FUNCTION F_DcToExt : T_DCTIME64  // Converts a DC time to a TAI-like absolute time expressed in T_DCTIME64 format.
VAR_INPUT
	dcTime: T_DCTIME64;  // 64-bit DC time.
END_VAR
VAR
END_VAR

F_DcToExt := F_ConvTcTimeToExtTime64(
	dcTime,
	LINT_TO_ULINT(GVL.DcToTcTimeOffset),
	LINT_TO_ULINT(GVL.DcToExtTimeOffset)
);

END_FUNCTION

(* stored: Version 1.1.0.1, ProductVersion 3.1.4022.18
   POU F_DcToExt: Id {87a0d92f-e837-404c-80d3-8113dc33c225}, SpecialFunc None *)
